PROGRAM PRG_OPT_SLITS
VAR
	fbSlits_Opt: FB_Slits;
	bExecuteMotion: BOOL := TRUE;
	bMoveOk: BOOL :=TRUE;
	bInit:BOOl:=TRUE;
END_VAR

// 4 jaws slit

IF bInit THEN
	bInit := FALSE;
	
	GVL_Main.M3.nBrakeMode := ENUM_StageBrakeMode.NO_BRAKE;
	GVL_Main.M3.bHardwareEnable := TRUE;
	GVL_Main.M3.bPowerSelf := TRUE;
	
	GVL_Main.M4.nBrakeMode := ENUM_StageBrakeMode.NO_BRAKE;
	GVL_Main.M4.bHardwareEnable := TRUE;
	GVL_Main.M4.bPowerSelf := TRUE;
	GVL_Main.M5.nBrakeMode := ENUM_StageBrakeMode.NO_BRAKE;
	GVL_Main.M5.bHardwareEnable := TRUE;
	GVL_Main.M5.bPowerSelf := TRUE;
	GVL_Main.M6.nBrakeMode := ENUM_StageBrakeMode.NO_BRAKE;
	GVL_Main.M6.bHardwareEnable := TRUE;
	GVL_Main.M6.bPowerSelf := TRUE;
	
	
	//
	GVL_Main.M3.nEnableMode := ENUM_StageEnableMode.DURING_MOTION ;
	GVL_Main.M4.nEnableMode := ENUM_StageEnableMode.DURING_MOTION ;
	GVL_Main.M5.nEnableMode := ENUM_StageEnableMode.DURING_MOTION ;
	GVL_Main.M6.nEnableMode := ENUM_StageEnableMode.DURING_MOTION ;
END_IF



fbSlits_Opt(	i_DevName:=					'OPT_SLITS',
				stTopBlade:=				GVL_Main.M5,
				stBottomBlade:=				GVL_Main.M6,
				stLeftBlade:=				GVL_Main.M3,
				stRightBlade:=				GVL_Main.M4,
				io_fbFFHWO:=				GVL_PMPS.io_fbFFHWO,
				fbArbiter:=					GVL_PMPS.fbArbiter,
				bExecuteMotion:=			bExecuteMotion,
				bMoveOk:=					bMoveOk
);

END_PROGRAM

(* stored: Version 1.1.0.1, ProductVersion 3.1.4022.18
   POU PRG_OPT_SLITS: Id {87d69d5e-6db8-4f14-b5ec-7224a0a8195a}, SpecialFunc None *)
